FUNCTION_BLOCK FCCStimuli
  (* Version 1.0, 2006-08-23, Goran Cengic, Chalmers *)
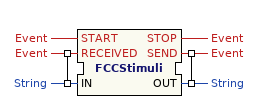
  EVENT_INPUT
    START;
    RECEIVED WITH IN;
  END_EVENT
  EVENT_OUTPUT
    STOP;
    SEND WITH OUT;
  END_EVENT
  VAR_INPUT
    IN : String;
  END_VAR
  VAR_OUTPUT
    OUT : String;
  END_VAR
  VAR
    time : DOUBLE;
  END_VAR
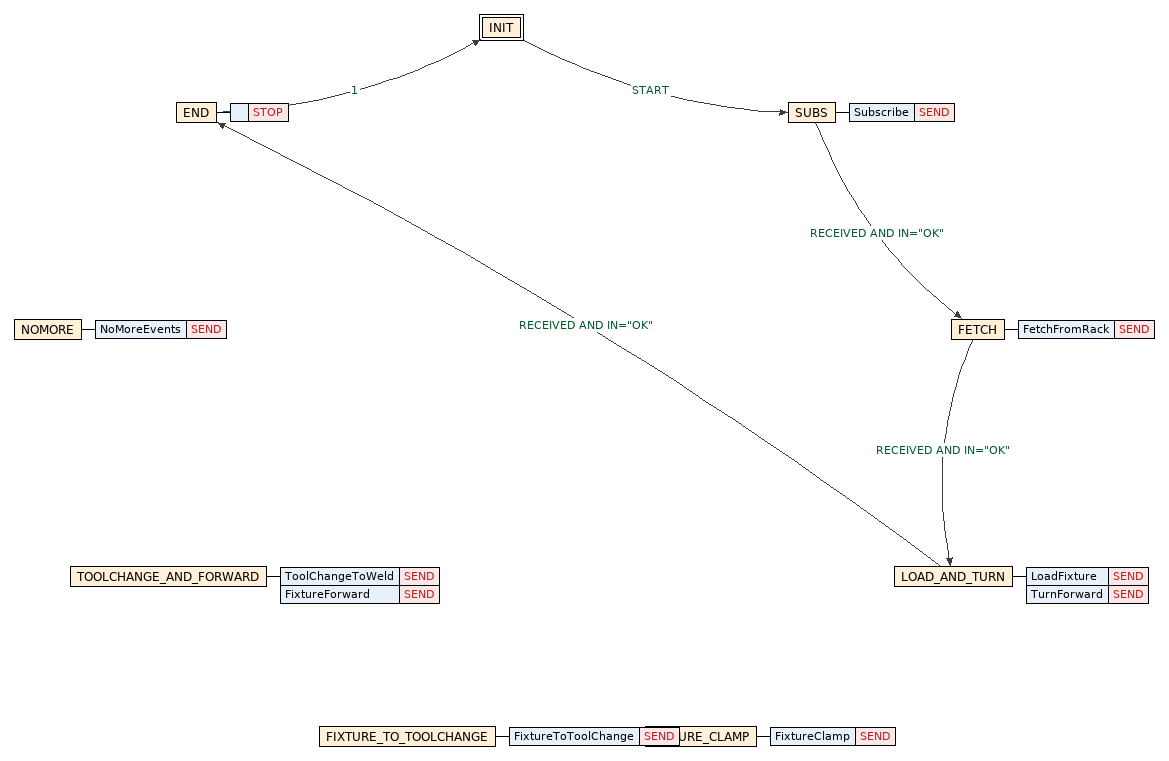
  EC_STATES
    INIT;
    SUBS : Subscribe -> SEND;
    FETCH : FetchFromRack -> SEND;
    LOAD_AND_TURN : LoadFixture -> SEND, TurnForward -> SEND;
    FIXTURE_CLAMP : FixtureClamp -> SEND;
    FIXTURE_TO_TOOLCHANGE : FixtureToToolChange -> SEND;
    TOOLCHANGE_AND_FORWARD : ToolChangeToWeld -> SEND, FixtureForward -> SEND;
    NOMORE : NoMoreEvents -> SEND;
    END : -> STOP;
  END_STATES
  EC_TRANSITIONS
    INIT TO SUBS := START;
    SUBS TO FETCH := RECEIVED AND IN="OK";
    FETCH TO LOAD_AND_TURN := RECEIVED AND IN="OK";
    LOAD_AND_TURN TO END := RECEIVED AND IN="OK";
    END TO INIT := 1;
  END_TRANSITIONS
  ALGORITHM Subscribe IN Java:
	 OUT = "SUBSCRIBE FetchFromRackf, LoadFixturef, FixtureClampf";
  END_ALGORITHM
  ALGORITHM Start1 IN Java:
	 OUT = "START FetchFromRacks 0";
  END_ALGORITHM
  ALGORITHM NoMoreEvents IN Java:
	 OUT = "NOMOREEVENTS";
  END_ALGORITHM
  ALGORITHM GetTime IN Java:

  END_ALGORITHM
END_FUNCTION_BLOCK
